{attribute 'linkalways'} 
{attribute 'no_explicit_call' := 'This FB is a CLASS and must be accessed using methods or properties'}
{attribute 'enable_dynamic_creation'}
FUNCTION_BLOCK Node_F_VN_FillContainer_ULINT EXTENDS VisionNode
VAR
    ipContainer : _ITcVnContainer;
    nValue : _ULINT(0);
    hrPrev : _HRESULT(S_OK);
    hresult : _HRESULT(S_OK);
END_VAR

METHOD PUBLIC  Clone : I_Node
VAR
    pNode : POINTER TO Node_F_VN_FillContainer_ULINT;
END_VAR
pNode := __NEW(Node_F_VN_FillContainer_ULINT);
Clone := pNode^;
END_METHOD

METHOD FB_init : BOOL
VAR_INPUT
    bInitRetains : BOOL; // if TRUE, the retain variables are initialized (warm start / cold start)
    bInCopyCode : BOOL;  // if TRUE, the instance afterwards gets moved into the copy code (online change)
END_VAR
AddInput('ipContainer', ipContainer);
AddInput('nValue', nValue);
AddInput('hrPrev', hrPrev);
AddOutput('ipContainer', ipContainer);
AddOutput('hresult',hresult);
END_METHOD

METHOD PROTECTED OnExecute : HRESULT
hresult.Value := F_VN_FillContainer_ULINT(
    ipContainer := ipContainer.Value,
    nValue := nValue.Value,
    hrPrev:= hrPrev.Value);
END_METHOD

METHOD PUBLIC PreExecutionCheck
VAR_INPUT
    Check : I_PreExecutionChecks;
END_VAR
Check.IsTrue(ipContainer.IsValid, 'ipContainer must be a valid container');
END_METHOD

END_FUNCTION_BLOCK

(* stored: Version 1.1.0.1, ProductVersion 3.1.4024.13
   POU Node_F_VN_FillContainer_ULINT: Id {253d9e91-6835-4cb6-b046-e8ba7cf00ddd}, SpecialFunc None
   Folder Constructor: Id {551a4e2c-c161-4faa-aa63-fee974405853}
   Method Clone: Id {8132e897-09c4-4772-845a-c0d53eed9087}
   Method FB_init: Id {8852689f-32b8-41c3-a2f6-7b48fdf66d18}
   Method OnExecute: Id {08b7ccc6-ee78-48bb-bad5-fe04fda02310}
   Method PreExecutionCheck: Id {2e78d80c-7869-461c-a8b2-f0445947c584} *)
